(* IEC 61131-3 sources: windowtracking/src/Others, 5 files *)

(* ---- IExitPointHandler.st ---- *)
NAMESPACE Simatic.Ax.WindowTracking.ExitPointHandler
    INTERFACE IExitPointHandler
        METHOD IsReady : BOOL
        END_METHOD

        METHOD Activate : BOOL
        END_METHOD

    END_INTERFACE
END_NAMESPACE

(* ---- ISortDecission.st ---- *)
USING Simatic.Ax.WindowTracking.Trigger;
USING Simatic.Ax.WindowTracking.ExitPointHandler;

NAMESPACE Simatic.Ax.WindowTracking.SortDecission
    INTERFACE ISortDecission
        METHOD Check : BOOL
            VAR_INPUT
                tw : ITransportWindow;
                te : IVirtualTrigger;
                exitpoint : IExitPointHandler;
            END_VAR
        END_METHOD
    END_INTERFACE
END_NAMESPACE

(* ---- ISortStrategy.st ---- *)
USING Simatic.Ax.WindowTracking.Trigger;
USING Simatic.Ax.WindowTracking.ExitPointHandler;

NAMESPACE Simatic.Ax.WindowTracking.SortDecission
    INTERFACE ISortStrategy
        METHOD Check : BOOL
            VAR_INPUT
                tw : ITransportWindow;
                te : IVirtualTrigger;
                exitpoint : IExitPointHandler;
            END_VAR
        END_METHOD
    END_INTERFACE
END_NAMESPACE

(* ---- SortDecisionOneDestination.st ---- *)
NAMESPACE Simatic.Ax.WindowTracking
    CLASS SortDecisionOneDestination IMPLEMENTS ISortStrategy
        VAR PUBLIC

        END_VAR
        VAR PROTECTED

        END_VAR

        METHOD PUBLIC Check : BOOL
            VAR_INPUT
                tw : ITransportWindow;
                te : IVirtualTrigger;
                exitpoint : IExitPointHandler;
            END_VAR
            VAR_TEMP
                _item : REF_TO ItemOneDestination;
            END_VAR
            _item ?= tw.GetItem();
            IF (_item = NULL) THEN
                Check := FALSE;
                RETURN;
            END_IF;
            IF (NOT exitpoint.IsReady()) THEN
                Check := FALSE;
                RETURN;
            END_IF;
            IF (_item^.GetDestination() = te) THEN
                Check := TRUE;
                RETURN;
            END_IF;
        END_METHOD
    END_CLASS
END_NAMESPACE

(* ---- SortDecissionOneDestination.st ---- *)
USING Simatic.Ax.WindowTracking.Items;
USING Simatic.Ax.WindowTracking.Trigger;
USING Simatic.Ax.WindowTracking.ExitPointHandler;

NAMESPACE Simatic.Ax.WindowTracking.SortDecission
    CLASS SortDecissionOneDestination IMPLEMENTS ISortDecission
        VAR PUBLIC

        END_VAR
        VAR PROTECTED

        END_VAR

        METHOD PUBLIC Check : BOOL
            VAR_INPUT
                tw : ITransportWindow;
                te : IVirtualTrigger;
                exitpoint : IExitPointHandler;
            END_VAR
            VAR_TEMP
                _item : REF_TO ItemOneDestination;
            END_VAR
            _item ?= tw.GetItem();
            IF (_item = NULL) THEN
                Check := FALSE;
                RETURN;
            END_IF;
            IF (NOT exitpoint.IsReady()) THEN
                Check := FALSE;
                RETURN;
            END_IF;
            IF (_item^.GetDestination() = te) THEN
                Check := TRUE;
                RETURN;
            END_IF;
        END_METHOD
    END_CLASS
END_NAMESPACE
